{attribute 'strict'}
TYPE E_CR800StateCyclePausing :
(
	CR800_CYCLE_PAUSING_IDLE	:= 0,	(* DUMMY *)
	CR800_CYCLE_PAUSING			:= 10,	(* Pausing in opearation *)
	CR800_CYCLE_PAUSING_DONE	:= 30	(* Pausing done *)
); 
END_TYPE

(* stored: Version 1.1.0.1, ProductVersion 3.1.4024.12
   DUT E_CR800StateCyclePausing: Id {cc0d7e26-9779-4dab-8ce0-e420c58006c3} *)
